TYPE DUT_SERVER_SKILL_INPUT :
STRUCT
	///Range of parameters
	ParameterInput: DUT_SERVER_PARAMETERINPUTARRAY;
	///Start process
	Execute: BOOL;
END_STRUCT
END_TYPE

(* stored: Version 1.1.0.1, ProductVersion 3.1.0.25
   DUT DUT_SERVER_SKILL_INPUT: Id {b3bc7e6b-4af7-49a9-af6b-49f8eea15794} *)
